// TwinCAT 3 PLC project PLC
// ProgramVersion: 3.1.4023.0
// libraries:
//   Tc2_EtherCAT, * (Beckhoff Automation GmbH)
//   Tc2_Standard, * (Beckhoff Automation GmbH)
//   Tc2_System, * (Beckhoff Automation GmbH)
//   Tc3_EventLogger, * (Beckhoff Automation GmbH)
//   Tc3_Module, * (Beckhoff Automation GmbH)
// project tree:
//   / E_MainStateMachine.TcDUT, FB_CaseStateMachine.TcPOU, MAIN.TcPOU, PlcTask.TcTTO
// real-time tasks:
//   TASK PlcTask: cycle T#10ms, priority 20, ADS port 350

CONFIGURATION PLC
    RESOURCE PLC ON TwinCAT3
        TASK PlcTask(INTERVAL := T#10ms, PRIORITY := 20);
        PROGRAM MAIN WITH PlcTask : MAIN;
    END_RESOURCE
END_CONFIGURATION

// ---- E_MainStateMachine.TcDUT
{attribute 'qualified_only'}
{attribute 'strict'}
{attribute 'to_string'}
TYPE E_MainStateMachine :
(
	Init := 0,
    step0,
    step1,
    step2,
    step3,
    step4,
    TipStep,
    error
);
END_TYPE

// ---- MAIN.TcPOU
PROGRAM MAIN
VAR
    // state machine
    eState : E_MainStateMachine;
    (*The FB_Init method is used to pass the name of the state machine, the event entry and the variable of the state machine*)
    fbState : FB_CaseStateMachine('MainStateMachine', TC_Events.TcGeneralAdsEventClass.Pending,eState);

    //some transitions
    bInitDone : BOOL;
    bDoStuff : BOOL;
    timertrans1 : TON;
    nCount : INT;
    i : INT;

    //Error
    bError : BOOL;

    //TipMode
    bEnableTipMode : BOOL;  
    bTip : BOOL;   
END_VAR

(*With the following method, you can switch on the Tip Mode and define the appropriate step.*)
fbState.EnableTipMode(bEnable := bEnableTipMode, nTipModeState := E_MainStateMachine.TipStep);

(*the case statement is in a repeat loop. If the state is to be changed in the same cycle,
the repeat loop executes the case statement a second time. Be careful when using this function*)
REPEAT

    (*Instead of using an initiger or enum with the Case statement,
      the CyclicCase statement is executed. This is used to pass the step name.*)
    CASE fbState.CyclicCase(TO_STRING(eState)) OF
        E_MainStateMachine.Init:
            
            (*As with a traditional state machine, the state variable can be written to directly*)
            IF bInitDone THEN
                eState := E_MainStateMachine.step0;
                bInitDone := FALSE;
            END_IF
            IF bDoStuff THEN
                eState := E_MainStateMachine.step4;
                bDoStuff := FALSE;
            END_IF
    
        E_MainStateMachine.step0:
            (*Many operations do not have to be performed cyclically.
              The EntryStep and Exit Step properties can be read for this purpose.*)
            IF fbState.EntryStep THEN
                timertrans1.IN := TRUE;
                timertrans1.PT := T#5S;
            END_IF
    
            timertrans1();
            (*Instead of writing an If statement and writing directly to the state variable,
              the TransChangeStep method can be used. When the transition becomes true, the state is changed.*)
              
            fbState.TransChangeState(E_MainStateMachine.step1, timertrans1.Q);
            
            fbState.TransChangeState(E_MainStateMachine.error, bError);
            
            (*Send events for diagnostic purposes*)
            fbState.TransSendEvent(sText :='Ups, an error has occurred', sExtendsSourceInfo := '', bTransition := bError);
            
            IF fbState.ExitStep THEN
                timertrans1(IN := FALSE);
            END_IF
    
        E_MainStateMachine.step1:
   
            IF fbState.EntryStep THEN //entry step
               nCount := 0;
            END_IF
    
            //do Stuff
            FOR i := 0 TO 10 DO
                nCount := nCount + 1;
            END_FOR
            
            (*Instead of writing an If statement and writing the state variable directly,
            the ChangeStep method can be used to exit the state directly*)
            fbState.ChangeState(E_MainStateMachine.step2);
    
            IF fbState.ExitStep THEN //exit step
                nCount := 0;
            END_IF 
    
        E_MainStateMachine.step2:
        
            (*Some steps are just for organization or preparation.
              You can leave these steps and switch to another one in the same cycle.
              For this purpose you can use the mehode TransChangeStateAndRepeat.*)
            fbState.TransChangeStateAndRepeat(E_MainStateMachine.step3, TRUE);
           
        E_MainStateMachine.step3:
               
            (*do things and repeat the case statement in the same cycle*)
            IF bDoStuff THEN
                fbState.ChangeStateAndRepeat(E_MainStateMachine.step4);
                bDoStuff := FALSE;
            END_IF
            (*Some steps must be executed an exact time.
              Instead of creating TON function blocks you can use the property t.*)
            fbState.TransChangeState(E_MainStateMachine.Init, fbState.t >= T#5S);
            
        E_MainStateMachine.step4:
        
            (*get things done and return to the previous step*)
            fbState.TransChangeState(fbState.PreviousStep, fbState.t >= T#3S);    
        
        E_MainStateMachine.error:
    
            fbState.TransChangeState(E_MainStateMachine.Init, NOT bError);
            
        E_MainStateMachine.TipStep :
        
            fbState.TipModeAllowNextStep(bTip);
            bTip := FALSE;
        ELSE
            (*Always use an Else branch in case something does go wrong ;)

            Todo : Perform error handling here*)
            fbState.ChangeState(E_MainStateMachine.Init);
    END_CASE
    
 (*This checks whether the case statement needs to be executed again.
   Unfortunately there is an error in the compiler which makes it necessary to add an "And True".
   Otherwise no Brakepoints are possible.*)   
UNTIL fbState.NotToBeRepeated AND TRUE END_REPEAT

END_PROGRAM

// ---- FB_CaseStateMachine.TcPOU
(*

enum : E_AnyEnum;
fb : FB_StepState('Name',TC_Evetns.Eventclass.Event,enum);

Use the method as Case Variable ->
CASE fb.CyclicCaseOf(TO_String(enum)) OF
1: ;
2: ;
IF fb.EntryStep THEN
; // Do Stuff
END_IF

ELSE ;
END_CASE

and use the property "State" as your Case variable. Then they can request the property "EntryState" in their step sequence to request the first execution of the step.*)
{attribute 'no_explicit_call' := 'do not call this POU directly'}
FUNCTION_BLOCK FB_CaseStateMachine
VAR
    {attribute 'hide'}
    nState : REFERENCE TO INT; //current state
    {attribute 'hide'}
    nNextStep : INT; //current state
    {attribute 'hide'}
    nStateTemp : INT;
    {attribute 'hide'}
    bEntryStep : BOOL; //the current state is called the first time
    {attribute 'hide'}
    EventEntry : TcEventEntry;
    {attribute 'hide'}
    sNameOfTheStateMachine : Tc2_System.T_MaxString; //name of the state machine
    {attribute 'hide'}
    sState : Tc2_System.T_MaxString; //name of the current state
    {attribute 'hide'}
    nStateAtBeginning : INT; //state of the Beginning of the Cycle
    {attribute 'hide'}
    nPreviousState : INT; //previous state
    {attribute 'hide'}
    sPreviousState : Tc2_System.T_MaxString;//name of the previous state
    {attribute 'hide'}
    bToBeRepeated : BOOL; //case instruction should be repeated in the same cycle
    {attribute 'hide'}
    CycleStarted : ULINT; //time when the current condition occurred for the first time
    {attribute 'hide'}
    bEnabledTipMode : BOOL;
    {attribute 'hide'}
    nTipModeState : INT;
END_VAR

//change the current state
METHOD PUBLIC ChangeState : HRESULT
VAR_INPUT
    nState : INT;
END_VAR
ChangeState := S_OK;
THIS^.nNextStep := nState;
bToBeRepeated := FALSE; //dont repeat the case statement
TipModeLogic();
END_METHOD

//change the current state and repeat the case statement in the same cycle.
METHOD PUBLIC ChangeStateAndRepeat : HRESULT
VAR_INPUT
    nState : INT;
END_VAR
ChangeStateAndRepeat := S_OK;
THIS^.nNextStep := nState;
bToBeRepeated := TRUE; //Repeat the case statement
TipModeLogic();
END_METHOD

(*
Use the method as Case Variable ->
CASE fb.CyclicCaseOf(TO_String(enum)) OF
1: ;
2: ;
ELSE ;
END_CASE
*)

{attribute 'monitoring':='variable'}
METHOD PUBLIC CyclicCase : INT
VAR_INPUT
    sState : Tc2_System.T_MaxString;//Name of the current state (TO_String(enum))
END_VAR
VAR_INST
    bInit : BOOL := TRUE;
END_VAR
bEntryStep := (nStateTemp <> nState) OR bInit; //check for change to recognize the entry step
bToBeRepeated := FALSE; //reset the ToBeRepeated flag

IF bEntryStep THEN

    
    // Save PreviousState
    IF bInit THEN
        nPreviousState := nState;
        sPreviousState := sState;
    ELSE
        nPreviousState := nStateTemp;
        sPreviousState := THIS^.sState;
	END_IF
    
    // Save active State
    nStateTemp := nState;
    THIS^.sState := sState; //save aktive state string
    Logging(); //Logging after the new state has been adopted
    bInit := FALSE;
    CycleStarted := F_GetActualDcTime64(); // Save timestamp   
END_IF

CyclicCase := nState; //return state
nStateAtBeginning := nState; //save the state at the beginning
END_METHOD

METHOD PUBLIC EnableTipMode : HRESULT
VAR_INPUT
    bEnable : BOOL;
    nTipModeState : INT; //The state to jump to when the step chain is in TipMode.
END_VAR
THIS^.bEnabledTipMode := bEnable;
THIS^.nTipModeState := nTipModeState;
END_METHOD

{attribute 'monitoring':='variable'}
//the current state is called the first time
PROPERTY PUBLIC EntryStep : BOOL
GET
EntryStep := bEntryStep;
END_GET
END_PROPERTY

//the current state is exited now
PROPERTY PUBLIC ExitStep : BOOL
GET
ExitStep := nStateAtBeginning <> nState;
END_GET
END_PROPERTY

METHOD FB_init : BOOL
VAR_INPUT
    bInitRetains : BOOL; // if TRUE, the retain variables are initialized (warm start / cold start)
    bInCopyCode : BOOL; // if TRUE, the instance afterwards gets moved into the copy code (online change)
    sNameOfTheStateMachine : Tc2_System.T_MaxString; //Name of the state machine
    EventEntry : TcEventEntry; //TwinCAT3 event entry
    EnumRef : REFERENCE TO INT; //Reference to an enum which represents the states of the state machine.    
END_VAR
THIS^.sNameOfTheStateMachine := sNameOfTheStateMachine;
THIS^.EventEntry := EventEntry;
THIS^.nState REF= EnumRef;
THIS^.nNextStep := nState;
END_METHOD

METHOD PROTECTED Logging : HRESULT
VAR
    sText : T_MaxString;
    sOldTime : T_MaxString;
END_VAR
VAR_INST
    {attribute 'tc_no_symbol'}
    {attribute 'hide'}
    fbMessage : FB_TcMessage;
    {attribute 'no_copy'}
    fbSourceInfo : FB_TcSourceInfo;
    bInit : BOOL := TRUE;
    sDifTime : STRING;
END_VAR
IF bInit THEN
    fbSourceInfo.ResetToDefault();
    fbMessage.CreateEx(EventEntry, fbSourceInfo);    
    bInit := FALSE;
END_IF

sText := CONCAT('StateMachine: ', (CONCAT(sNameOfTheStateMachine, CONCAT(', State: ', StateAsString)))); //name of the current step

IF CycleStarted <> 0 THEN // Add last execution time
    sOldTime := CONCAT('[Last state: ', PreviousStepAsString); //name of the previous step
    sOldTime := CONCAT(sOldTime, '(');
    sDifTime := DELETE (LTIME_TO_STRING( ULINT_TO_LTIME(F_GetActualDcTime64() - CycleStarted)), 6,1);
    sOldTime := CONCAT(sOldTime, sDifTime);
    sOldTime := CONCAT(sOldTime, ')]');

    sText := CONCAT(sText, ' ');
    sText := CONCAT(sText, sOldTime);
END_IF
//Send Message
fbMessage.ipArguments.Clear().AddString(sText);
fbMessage.Send(nTimeStamp := 0);
END_METHOD

//Case instruction should NOT be repeated in the same cycle
PROPERTY PUBLIC NotToBeRepeated : BOOL
GET
NotToBeRepeated := NOT bToBeRepeated;
END_GET
END_PROPERTY

{attribute 'monitoring':='call'}
//previous state
PROPERTY PUBLIC PreviousStep : INT
GET
PreviousStep := nPreviousState;
END_GET
END_PROPERTY

{attribute 'monitoring':='call'}
//previous state as STRING
PROPERTY PUBLIC PreviousStepAsString : T_MaxString
GET
PreviousStepAsString := sPreviousState;
END_GET
END_PROPERTY

METHOD PUBLIC SendEvent : HRESULT
VAR_INPUT
	sText: STRING(255);
	sExtendsSourceInfo: STRING(255);
END_VAR
VAR_INST
    {attribute 'tc_no_symbol'}
    {attribute 'hide'}
    fbMessage : FB_TcMessage;
    {attribute 'no_copy'}
    fbSourceInfo : FB_TcSourceInfo;
    bInit : BOOL := TRUE;
END_VAR
IF bInit THEN
    fbSourceInfo.ResetToDefault();
    fbMessage.CreateEx(EventEntry, fbSourceInfo);    
    bInit := FALSE;
END_IF


IF sExtendsSourceInfo <> '' THEN    
    fbSourceInfo.ExtendName(sExtendsSourceInfo);
END_IF
    fbMessage.ipArguments.Clear().AddString(sText);
    fbMessage.Send(nTimeStamp := 0);

IF sExtendsSourceInfo <> '' THEN
    fbSourceInfo.ResetToDefault();
END_IF
END_METHOD

{attribute 'monitoring':='call'}
//current state
PROPERTY PUBLIC State : INT
GET
State := nState;
END_GET
END_PROPERTY

{attribute 'monitoring':='variable'}
//name of the current state
PROPERTY PUBLIC StateAsString : T_MaxString
GET
StateAsString := sState;
END_GET
END_PROPERTY

{attribute 'monitoring':='call'}
//Time spent in current state
PROPERTY PUBLIC t : TIME
GET
t := ULINT_TO_TIME((F_GetSystemTime() - CycleStarted) / 10000);
END_GET
END_PROPERTY

METHOD PUBLIC TipModeAllowNextStep : HRESULT
VAR_INPUT
    bTransition : BOOL;
END_VAR
IF bTransition THEN
    nState := nNextStep;       
END_IF
TipModeAllowNextStep := Tc3_Module.S_OK;
END_METHOD

METHOD PROTECTED TipModeLogic : HRESULT
VAR_INPUT
END_VAR
(*If TipMode is not active, the new step is applied immediately.*)
IF NOT bEnabledTipMode THEN
    nState := nNextStep;
ELSE
    nState := nTipModeState;
END_IF
TipModeLogic := Tc3_Module.S_OK;
END_METHOD

//change the current state as soon as the transition becomes TRUE
METHOD PUBLIC TransChangeState : HRESULT
VAR_INPUT
    nState : INT;
    bTransition : BOOL;
END_VAR
TransChangeState := S_PENDING;
IF bTransition THEN
    THIS^.nNextStep := nState;
    TransChangeState := S_OK;
    bToBeRepeated := FALSE; //dont repeat the case statement
    TipModeLogic();
END_IF
END_METHOD

//change the current state if the transition is true, and repeat the case statement in the same cycle.
METHOD TransChangeStateAndRepeat : HRESULT
VAR_INPUT
    nState : INT;
    bTransition : BOOL;
END_VAR
TransChangeStateAndRepeat := S_PENDING;
IF bTransition THEN
    THIS^.nNextStep := nState;
    TransChangeStateAndRepeat := S_OK;
    bToBeRepeated := TRUE; //Repeat the case statement
    TipModeLogic();
END_IF
END_METHOD

METHOD PUBLIC TransSendEvent : HRESULT
VAR_INPUT
	sText: STRING(255);
	sExtendsSourceInfo: STRING(255);
    bTransition : BOOL;
END_VAR
VAR_INST
    {attribute 'tc_no_symbol'}
    {attribute 'hide'}
    fbMessage : FB_TcMessage;
    {attribute 'no_copy'}
    fbSourceInfo : FB_TcSourceInfo;
    bInit : BOOL := TRUE;
END_VAR
IF bTransition THEN
    SendEvent(sExtendsSourceInfo := sExtendsSourceInfo, sText := sText);
END_IF
END_METHOD

END_FUNCTION_BLOCK
